PROGRAM PRG_DPL_X_EPS
VAR
    bInit 		: BOOL := TRUE;

    fDPL_X 		: LREAL;
    fSDS_RY 	: LREAL;
    fDPL_Z 		: LREAL;
    bFullRange 	: BOOL;

    fbEPS		: FB_EPS;

END_VAR

IF bInit THEN
    // Set Inital Values
    aDPL_X_EPS[1].fBwd_Limits := 10;
    aDPL_X_EPS[1].fFwd_Limits := 80;

    aDPL_X_EPS[2].fBwd_Limits := 10;
    aDPL_X_EPS[2].fFwd_Limits := 30;

    aDPL_X_EPS[3].fBwd_Limits := 30;
    aDPL_X_EPS[3].fFwd_Limits := 80;


    bInit := FALSE;
END_IF

fDPL_X  := M1.stAxisStatus.fActPosition;
fSDS_RY := M19.stAxisStatus.fActPosition;
fDPL_Z 	:= M3.stAxisStatus.fActPosition;


fbEPS(eps:=aDPL_X_EPS[2].stEPS);
fbEPS.setDescription('DPL_RY in [10,30]');
fbEPS.setBit(0, F_InRange(fSDS_RY, 10, 30));

fbEPS(eps:=aDPL_X_EPS[3].stEPS);
fbEPS.setDescription('DPL_Z in [10,30]');
fbEPS.setBit(0, F_InRange(fDPL_Z, 30, 80));

bFullRange := (NOT aDPL_X_EPS[2].stEPS.bEPS_OK) AND (NOT aDPL_X_EPS[3].stEPS.bEPS_OK);

fbEPS(eps:=aDPL_X_EPS[1].stEPS);
fbEPS.setDescription('Full Range');
fbEPS.setBit(0, bFullRange);

F_CheckEPSArray(stMotor:= M3, aEPSLimits:= aDPL_X_EPS, nStart:= 1, nEnd:= 3);

END_PROGRAM

(* stored: Version 1.1.0.1, ProductVersion 3.1.4022.18
   POU PRG_DPL_X_EPS: Id {04026f9f-33ec-468b-8c87-d293a0ccda10}, SpecialFunc None *)
